FUNCTION_BLOCK ABSTRACT Queue
VAR
	dataSize : ULINT; //no functionaility, only to force input a type for readability
	varType : __SYSTEM.TYPE_CLASS;
END_VAR
VAR
	elements : FB_BA_DynamicArray := (uiEntrySize := 2, uiMinExpCount := GVL.initArraySize);
	length : USINT := 0;
	uiEntrySizeRef : REFERENCE TO UINT;
END_VAR

END_FUNCTION_BLOCK

(* stored: Version 1.1.0.1, ProductVersion 3.1.4024.11
   POU Queue: Id {cc03ee38-0c22-4ccc-9545-2ee091a456fb}, SpecialFunc None *)
